Yaskawa INFORM job: TRIAL2.JBI

/JOB
//NAME TRIAL2
//POS
///NPOS 14,0,0,0,0,0
///TOOL 0
///POSTYPE PULSE
///PULSE
C00000=-170684,-159276,70742,-9914,-117427,-102131
C00001=-163021,-158485,66126,-3704,-115003,-92973
C00002=-163555,-160727,60854,-4075,-113503,-93005
C00003=-163767,-162339,56863,-4201,-112327,-92987
C00004=-163059,-163014,54639,-3639,-111573,-92848
C00005=-160600,-158662,58178,-2741,-116641,-104659
C00006=-160911,-158936,57414,-2979,-116393,-104699
C00007=-149553,-160674,44203,5710,-110608,-103320
C00008=-159415,-161021,39321,24500,-110372,-99511
C00009=-169334,-166129,23462,44842,-103180,-97173
C00010=-171380,-170239,14903,49777,-100632,-97182
C00011=-202441,-174961,-27742,25505,-78055,-88420
C00012=-185981,-168812,-19506,525,-93918,-88112
C00013=-185981,-168812,-19506,525,-93918,-88112
//INST
///DATE 2022/04/06 10:57
///ATTR SC,RW
///GROUP1 RB1
NOP
MOVJ C00000 VJ=65.00
MOVL C00001 V=150.0
MOVC C00002 V=150.0
MOVC C00003 V=150.0
MOVC C00004 V=150.0
MOVL C00005 V=150.0
MOVL C00006 V=150.0
MOVL C00007 V=150.0
MOVL C00008 V=150.0
MOVL C00009 V=150.0
MOVL C00010 V=150.0
MOVL C00011 V=150.0
MOVL C00012 V=150.0
MOVJ C00013 VJ=65.00
END
